// TwinCAT 3 PLC project FirstPlcProject
// ProgramVersion: 3.1.4024.0
// libraries:
//   Tc2_Standard, * (Beckhoff Automation GmbH)
//   Tc2_System, * (Beckhoff Automation GmbH)
//   Tc3_Module, * (Beckhoff Automation GmbH)
// project tree:
//   / PlcTask.TcTTO
//   POUs/ MAIN.TcPOU

CONFIGURATION FirstPlcProject
    RESOURCE PLC ON TwinCAT3
        TASK PlcTask(INTERVAL := T#10ms, PRIORITY := 20);
        PROGRAM MAIN WITH PlcTask : MAIN;
    END_RESOURCE
END_CONFIGURATION

// ---- POUs/MAIN.TcPOU
// Deklarationsbereich

PROGRAM MAIN
VAR
	bIn1, bIn2, bOut : BOOL;
END_VAR

// Anweisungsbereich

bOut := bIn1 AND bIn2;		//Logisches AND

(*
Comment for multiple lines
*)

END_PROGRAM
